{attribute 'c++_compatible'}
FUNCTION_BLOCK TransportSystemSlave EXTENDS TcBaseModuleRegistered IMPLEMENTS I_TransportSlave
VAR_INPUT
END_VAR
VAR_OUTPUT
END_VAR
VAR
(*
Naive Implementierung um MC_GearInVelo / GearOut nachzubilden.
*)

	// ==== Motion Control ====
	axisTransportB: AXIS_REF;		// Slave
	
	// ==== Inputs =====
	rMasterVelocity AT %I*: LREAL;	// Master velocity
	
END_VAR

axisTransportB.ReadStatus();

METHOD FB_reinit : BOOL
VAR_INPUT
END_VAR
SUPER^.FB_reinit();
END_METHOD

{attribute 'TcTypeSystem'}
{attribute 'no-analysis'}
{attribute 'c++_compatible'}
{attribute 'minimal_input_size' := '4'}
{attribute 'pack_mode' := '4'}
{warning 'Methodenimplementierung hinzufügen'}
(* Anhalten *)
METHOD Halt : HRESULT
END_METHOD

{attribute 'TcTypeSystem'}
{attribute 'no-analysis'}
{attribute 'c++_compatible'}
{attribute 'minimal_input_size' := '4'}
{attribute 'pack_mode' := '4'}
(* Passe dich der Master-Geschwindigkeit an *)
METHOD SyncWithMaster : HRESULT
END_METHOD

{attribute 'TcTypeSystem'}
{attribute 'no-analysis'}
{attribute 'c++_compatible'}
{attribute 'minimal_input_size' := '4'}
{attribute 'pack_mode' := '4'}
METHOD TcQueryInterface : HRESULT
VAR_INPUT
	iid	: REFERENCE TO IID;
	pipItf	: POINTER TO PVOID;
END_VAR
VAR
	ipTPS: I_TransportSlave;
END_VAR
IF GuidsEqual(ADR(iid), ADR(TC_GLOBAL_IID_LIST.IID_I_TransportSlave)) THEN
	ipTPS := THIS^;
	pipItf^ := ITCUNKNOWN_TO_PVOID(ipTPS);
	TcAddRef();
	TcQueryInterface := S_OK;
ELSE
	TcQueryInterface := SUPER^.TcQueryInterface(iid, pipItf);
END_IF
END_METHOD

END_FUNCTION_BLOCK

(* stored: Version 1.1.0.1, ProductVersion 3.1.4024.3
   POU TransportSystemSlave: Id {0da10745-a5b5-4172-8fc3-cd4b7c709a8e}, SpecialFunc None
   Method FB_reinit: Id {ca8ee805-4052-4df1-b645-2aab0bad467b}
   Method Halt: Id {858be294-6224-4fde-96ad-4f14d61a50e4}
   Method SyncWithMaster: Id {ca67a40d-038f-433c-97d3-099d74d3da29}
   Method TcQueryInterface: Id {1775d457-38d0-47c4-ba06-fc0da9d2dbd4} *)
